{attribute 'linkalways'} 
{attribute 'no_explicit_call' := 'This FB is a CLASS and must be accessed using methods or properties'}
{attribute 'enable_dynamic_creation'}
FUNCTION_BLOCK FINAL AnyInterfaceDisplayNode EXTENDS Node
VAR
	in : I_InterfaceDatatype;
	display : I_InterfaceDatatype;
END_VAR

METHOD PUBLIC Clone : I_Node
VAR
	pNode : POINTER TO AnyInterfaceDisplayNode;
END_VAR
pNode := __NEW(AnyInterfaceDisplayNode(Datatype := in));
Clone := pNode^;
END_METHOD

METHOD FB_exit : BOOL
VAR_INPUT
	bInCopyCode : BOOL; // if TRUE, the exit method is called for exiting an instance that is copied afterwards (online change).
END_VAR
IF bInCopyCode THEN
	RETURN;
END_IF

in.Dispose();
display.Dispose();
END_METHOD

METHOD FB_init : BOOL
VAR_INPUT
	bInitRetains : BOOL; // if TRUE, the retain variables are initialized (warm start / cold start)
	bInCopyCode : BOOL;  // if TRUE, the instance afterwards gets moved into the copy code (online change)
	Datatype : I_InterfaceDatatype;
END_VAR
Datatype.Clone().TryResolveAsInterfaceDatatype(THIS^.in);
Datatype.Clone().TryResolveAsInterfaceDatatype(THIS^.display);

AddInput('in', THIS^.in);
AddContent('display', THIS^.display);
END_METHOD

METHOD PROTECTED OnExecute : HRESULT
VAR
END_VAR
display.TryCopyContentFrom(in);
END_METHOD

END_FUNCTION_BLOCK

(* stored: Version 1.1.0.1, ProductVersion 3.1.4024.13
   POU AnyInterfaceDisplayNode: Id {bc39b922-3d83-0130-2b11-7bb0ac973d48}, SpecialFunc None
   Folder Constructor: Id {ecc6e8b9-3762-07d2-2a21-6d015e4a15f5}
   Folder Destructor: Id {45744eff-e2e7-061e-39b9-fc774905e918}
   Method Clone: Id {178d4b9f-f18e-07fb-3c25-e938c0c068a1}
   Method FB_exit: Id {e85702b0-9f4f-0abc-351a-5cfd9319eea2}
   Method FB_init: Id {8b70c3e1-ec65-0e9a-1cf9-28c44c7d7644}
   Method OnExecute: Id {2e98590f-2783-02b3-02ff-8cd80273456f} *)
